Yaskawa INFORM job: R2_W53-A3(90,180)(Z_REKI)AWOK.JBI

/JOB
//NAME R2_W53-A3(90,180)(Z_REKI)AWOK
///FOLDERNAME AWOK
//POS
///NPOS 29,29,0,2,0,0
///TOOL 0
///POSTYPE PULSE
///PULSE
C00000=123351,93172,10868,-1707,101249,3089
C00001=121638,101600,23101,7580,97824,11972
C00002=120902,75334,17452,11788,87744,15726
C00003=120849,79304,25274,11826,85034,15453
C00004=120828,81036,28580,11850,83915,15340
C00005=120832,80505,29096,11858,83337,15286
C00006=120828,81036,28580,11850,83915,15340
C00007=120210,78530,25627,12070,84516,15204
C00008=119679,80391,27915,12273,84145,15000
C00009=120847,79349,26633,11838,84237,15377
C00010=120514,81256,29247,11970,83667,15217
C00011=120994,83062,31482,11812,83171,15324
C00012=120514,81256,29247,11970,83667,15217
C00013=120532,79503,25915,11946,84790,15331
C00014=120578,75485,18039,11908,87509,15605
C00015=93954,88980,33985,18355,88530,24680
C00016=93954,87354,35318,18360,86955,24443
C00017=93543,87426,36071,18479,86645,24262
C00018=93950,87325,35353,18361,86921,24437
C00019=94241,84522,33111,18268,86803,24514
C00020=92552,102461,54968,24694,88355,17224
C00021=92749,116421,73764,29015,90990,10179
C00022=87912,133052,104101,47712,88680,9724
C00023=93941,82559,42870,56987,100292,10162
C00024=93940,83160,41093,57260,101081,10714
C00025=90210,89066,48455,57402,102410,9426
C00026=90210,98956,38196,60599,108518,14111
C00027=90210,98956,38196,60599,61779,14111
C00028=90211,98953,38197,60599,61783,14111
BC00000=197421,328329,1075174
BC00001=177517,269426,1075174
BC00002=168072,241477,1075175
BC00003=168072,241477,1075175
BC00004=168072,241477,1075175
BC00005=168072,241477,1075175
BC00006=168072,241477,1075175
BC00007=168072,241477,1075175
BC00008=168072,241477,1075175
BC00009=168072,241477,1075175
BC00010=168072,241477,1075175
BC00011=168072,241478,1075168
BC00012=168072,241477,1075175
BC00013=168072,241477,1075175
BC00014=168072,241477,1075175
BC00015=67462,238148,1075175
BC00016=69147,233756,1075175
BC00017=69569,232658,1075171
BC00018=69822,232000,1075175
BC00019=69822,232000,1075175
BC00020=69569,232658,1075168
BC00021=69569,232658,1075168
BC00022=69569,232657,1075164
BC00023=118851,203745,1075175
BC00024=123428,207990,1075175
BC00025=123428,207990,1075175
BC00026=123428,207990,1075175
BC00027=123428,207990,1075175
BC00028=123428,477103,1075172
///POSTYPE BASE
///RECTAN
///RCONF 0,0,0,0,0,0,0,0,0,0,0,0,0,0,0,0,0,0,0,0,0,0,0,0
P00006=0.222,-3.123,-1.508,0.0000,0.0000,0.0000
P00023=0.143,-0.036,0.682,0.0000,0.0000,0.0000
//INST
///DATE 2023/11/01 18:05
///ATTR SC,RW
///GROUP1 RB1,BS1
NOP
'r2_W53-A3(90,180)(z_reki)
'Path S1003
SFTOF
MOVJ C00000 BC00000 VJ=50.00
MOVJ C00001 BC00001 VJ=50.00
MOVJ C00002 BC00002 VJ=100.00
MOVL C00003 BC00003 V=400.0
MOVL C00004 BC00004 V=60.0
REFP 3 C00005 BC00005
CALL JOB:SEARCH-R1
SET P023 P006
SFTON P023
MOVL C00006 BC00006 V=60.0
MOVL C00007 BC00007 V=60.0
REFP 3 C00008 BC00008
CALL JOB:SEARCH-R1
SET P023 P006
SFTON P023
MOVL C00009 BC00009 V=60.0
MOVL C00010 BC00010 V=60.0
REFP 3 C00011 BC00011
CALL JOB:SEARCH-R1
SET P023 P006
SFTON P023
MOVL C00012 BC00012 V=60.0
MOVL C00013 BC00013 V=400.0
MOVL C00014 BC00014 V=1000.0
'Path W1004
SFTOF
SFTON P023
MOVJ C00015 BC00015 VJ=100.00
MOVL C00016 BC00016 V=400.0
MOVL C00017 BC00017 V=100.0 PL=0
REFP 1 C00018 BC00018
REFP 2 C00019 BC00019
MACRO1 MJ#(0) ARGF9
ARCON
MOVL C00020 BC00020 V=10.8
MOVL C00021 BC00021 V=10.8
MOVL C00022 BC00022 V=10.8
ARCOF
MOVL C00023 BC00023 V=400.0
MOVL C00024 BC00024 V=1000.0
SFTOF
MOVL C00025 BC00025 V=1000.0
MOVJ C00026 BC00026 VJ=50.00
MOVJ C00027 BC00027 VJ=50.00
MOVJ C00028 BC00028 VJ=50.00
END
